// TIA Portal project "LOGO! - S7-1200" (V11)

(* hardware
DEVICE "SIMATIC 1200-Station_1"  S71200.Device
   slot 0: "S7-1200 Baugruppenträger"  Rack  V1.0
   slot 1: "PLC_1"  CPU 1214C AC/DC/Rly  6ES7 214-1BE30-0XB0  V2.1
*)

// ===== PLC "PLC_1"  CPU 1214C AC/DC/Rly =====

VAR_GLOBAL   // PLC tag table "Standard-Variablentabelle"
   "Tag_1" AT %I0.2 : Bool;
   "Tag_2" AT %I0.7 : Bool;
   "Tag_3" AT %Q0.0 : Bool;
END_VAR

DATA_BLOCK "Datenbaustein_1"   // DB1
{ S7_Optimized_Access := 'FALSE' }
VERSION : 0.1
   VAR
      I1 : Bool;
      I2 : Bool;
      I3 : Bool;
      I4 : Bool;
      I5 : Bool;
      I6 : Bool;
      AI1 : Word;
      AI2 : Word;
      Q1 : Bool;
      Q2 : Bool;
      Q3 : Bool;
      Q4 : Bool;
   END_VAR
BEGIN
END_DATA_BLOCK

ORGANIZATION_BLOCK "Main"   // OB1, FBD, ProgramCycle
TITLE = "Main Program Sweep (Cycle)"
{ S7_Optimized_Access := 'FALSE' }
VERSION : 0.1
BEGIN

REGION Network 1
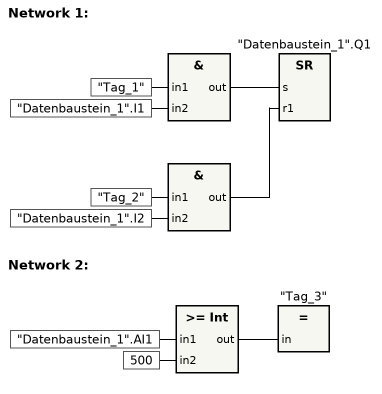
   IF "Tag_1" AND "Datenbaustein_1".I1 THEN
       "Datenbaustein_1".Q1 := TRUE;   // SR flip-flop
   END_IF;
   IF "Tag_2" AND "Datenbaustein_1".I2 THEN "Datenbaustein_1".Q1 := FALSE; END_IF;
END_REGION

REGION Network 2
   "Tag_3" := "Datenbaustein_1".AI1 >= 500;
END_REGION
END_ORGANIZATION_BLOCK